// TIA Portal V17 export
// export: Created 2025-03-05T08:02:28.3371619Z, ExportSetting WithDefaults, DisplayName Totally Integrated Automation Portal, DisplayVersion V17 Update 8, DisplayName TIA Portal Openness, DisplayVersion V17 Update 8, DisplayName TIA Portal Version Control Interface, DisplayVersion V17, DisplayName SINAMICS Startdrive Advanced, DisplayVersion V17 SP2, DisplayName SINAMICS Startdrive G110M, G120, G120C, G120D, G120P, G115D, DisplayVersion V17 SP2, DisplayName SINAMICS Startdrive G130, G150, S120, S150, SINAMICS MV, S210, DisplayVersion V17 SP2, DisplayName STEP 7 Professional, DisplayVersion V17 Update 8, DisplayName SINUMERIK ONE STEP 7 Toolbox, DisplayVersion V17 Update 12, DisplayName SINUMERIK 840D sl STEP 7 Toolbox, DisplayVersion V17 Update 12, DisplayName STEP 7 Safety, DisplayVersion V17 Update 6, DisplayName WinCC Advanced, DisplayVersion V17 Update 8
TYPE "LASER GUIDE"
// stored: IsFailsafeCompliant false
   STRUCT
      START_GENERAL_CONDITIONS : Bool;   // Start General Conditions
      START_GENERAL_CONDITIONS_HELP : Bool;   // Start General Conditions Help
      START_INITIAL_CONDITIONS : Bool;   // Start Initial Conditions
      START_INITIAL_CONDITIONS_HELP : Bool;   // Start Initial Conditions Help
      START_MANUAL_REQUEST : Bool;   // Start Manual Request
      FEEDBACK_ON : Bool;   // Feedback On
      START_AUTO_REQUEST : Bool;   // Start Auto Request
      START_GLOBAL_REQUEST : Bool;   // Start Global Request
      START_COMMAND : Bool;   // Start Command
      LASER_ON : Bool;   // Laser On
      STOP_GENERAL_CONDITIONS : Bool;   // Stop General Conditions
      STOP_GENERAL_CONDITIONS_HELP : Bool;   // Stop General Conditions Help
      STOP_INITIAL_CONDITIONS : Bool;   // Stop Initial Conditions
      STOP_INITIAL_CONDITIONS_HELP : Bool;   // Stop Initial Conditions Help
      STOP_MANUAL_REQUEST : Bool;   // Manual Stop Request
      STOP_AUTO_REQUEST : Bool;   // Auto Stop Request
      STOP_GLOBAL_REQUEST : Bool;   // Stop Global Request
      STOP_COMMAND : Bool;   // Stop Command
      STOPPED : Bool;   // Stopped
      FEEDBACK_OFF : Bool;   // Feedback Off
      LASER_FAULT : Bool;   // Laser Faulted
   END_STRUCT;
END_TYPE
